VISUALIZATION VISU_ST150  // 400x600
END_VISUALIZATION

(* stored: Version 1.1.0.1, ProductVersion 3.1.4024.6
   Visu VISU_ST150: Id {e3b53aa0-20d2-457e-acb8-c72d6d9848ef} *)
